PROGRAM Manual_Test
VAR
	FB_Servo : FB_RC_Servo;
	errorString : STRING;
	output : INT;
	stop : BOOL;
END_VAR

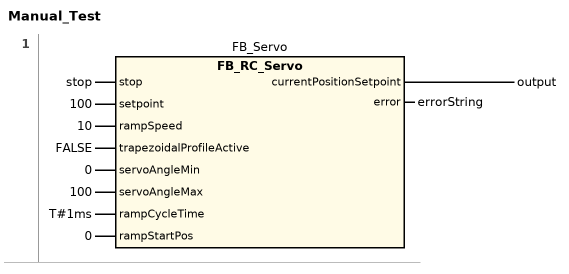
// NETWORK 1
FB_Servo(
    stop := stop,
    setpoint := 100,
    rampSpeed := 10,
    trapezoidalProfileActive := FALSE,
    servoAngleMin := 0,
    servoAngleMax := 100,
    rampCycleTime := T#1ms,
    rampStartPos := 0,
    error => errorString); // FB_RC_Servo
output := FB_Servo.currentPositionSetpoint;

END_PROGRAM

(* stored: Version 1.1.0.1, ProductVersion 3.1.4024.13
   POU Manual_Test: Id {21983412-0551-4a30-893d-729f040974d2}, SpecialFunc None *)
